// Mitsubishi GX Works2 project: group4TheoryB   PLC: FX3G

// global labels: Global1
VAR_GLOBAL
  StartSystem AT X010 : BOOL;
  SystemOn AT M0 : BOOL;
  SenOpen AT X003 : BOOL;
  SenDist AT X001 : BOOL;
  OpenGate AT Y001 : BOOL;
  SenClose AT X002 : BOOL;
  Open12Seconds AT TS1 : BOOL;
  CloseGate AT Y002 : BOOL;
END_VAR

// task Task_01 (event TRUE, interval 0, priority 31): POU_01

PROGRAM POU_01
(* structured ladder/FBD written out as ST: instructions are called as NAME(EN, inputs, outputs); _pN, _eN, _tN stand for wires *)
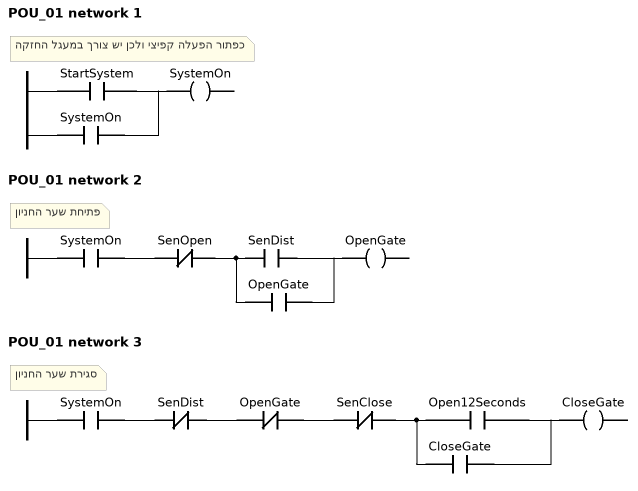
(* network 1 *)
(* כפתור הפעלה קפיצי ולכן יש צורך במעגל החזקה *)
SystemOn := StartSystem OR SystemOn;
(* network 2 *)
(* פתיחת שער החניון *)
_p1 := SystemOn AND NOT SenOpen;
OpenGate := (_p1 AND SenDist) OR (_p1 AND OpenGate);
(* network 3 *)
(* סגירת שער החניון *)
_p1 := SystemOn AND NOT SenDist AND NOT OpenGate AND NOT SenClose;
CloseGate := (_p1 AND Open12Seconds) OR (_p1 AND CloseGate);
END_PROGRAM
